PROGRAM MAIN
VAR
END_VAR

END_PROGRAM

(* stored: Version 1.1.0.1
   POU MAIN: Id {a3fd4a15-3d71-481c-b5ac-3fa459eb17e5} *)
